// TIA Portal V20 export
TYPE "typeSequenceControlNode"
// stored: Namespace Unit1.Em12
   STRUCT
      jobs : "LAF_typeJobs";
      sequence : "LAF_typeSequence";
      selectJobStatus { S7_SetPoint := 'True'} : Array[0..10] of "LAF_typeJobStatus";
      "step" : "LER_typeStep";
      jobInterface : "Unit1.Em12.typeSequenceControlNodeJobInterface";
      homeCheck : "Unit1.Em12.typeSequenceControlNodeHomeCheck";
   END_STRUCT;
   // // "step".action1[101] : Step[101] : JOB[1] Condition
   // // "step".action1[110] : Step[110] : Clamp Z Up
   // // "step".action1[120] : Step[120] : Clamp Left, Right Open
   // // "step".action1[130] : Step[130] : Clamp Mover Open
   // // "step".action1[180] : Step[180] : Lift Down
   // // "step".action1[190] : Step[190] : JOB[1] Step End
   // // "step".action1[201] : Step[201] : JOB[2] Condition
   // // "step".action1[210] : Step[210] : Stack NG Box [Loading Request] => JR Unloading P&P
   // // "step".action1[220] : Step[220] : Clamp Mover Close
   // // "step".action1[230] : Step[230] : Clamp Left, Right Close
   // // "step".action1[231] : Step[231] : Stack NG Box [Loading Ready] => JR Unloading P&P
   // // "step".action1[290] : Step[290] : JOB[2] Step End
   // // "step".action1[301] : Step[301] : JOB[3] Condition
   // // "step".action1[310] : Step[310] : Clamp Z Down
   // // "step".action1[320] : Step[320] : Clamp Left, Right Open
   // // "step".action1[330] : Step[330] : Clamp Mover Open
   // // "step".action1[340] : Step[340] : Clamp Z Up
   // // "step".action1[390] : Step[390] : JOB[3] Step End
   // // "step".transition1[101] : Step[101] : JOB[1] Condition
   // // "step".transition1[110] : Step[110] : Clamp Z Up
   // // "step".transition1[120] : Step[120] : Clamp Left, Right Open
   // // "step".transition1[130] : Step[130] : Clamp Mover Open
   // // "step".transition1[180] : Step[180] : Lift Down
   // // "step".transition1[190] : Step[190] : JOB[1] Step End
   // // "step".transition1[201] : Step[201] : JOB[2] Condition
   // // "step".transition1[210] : Step[210] : Stack NG Box [Loading Request] => JR Unloading P&P
   // // "step".transition1[220] : Step[220] : Clamp Mover Close
   // // "step".transition1[230] : Step[230] : Clamp Left, Right Close
   // // "step".transition1[231] : Step[231] : Stack NG Box [Loading Ready] => JR Unloading P&P
   // // "step".transition1[290] : Step[290] : JOB[2] Step End
   // // "step".transition1[301] : Step[301] : JOB[3] Condition
   // // "step".transition1[310] : Step[310] : Clamp Z Down
   // // "step".transition1[320] : Step[320] : Clamp Left, Right Open
   // // "step".transition1[330] : Step[330] : Clamp Mover Open
   // // "step".transition1[340] : Step[340] : Clamp Z Up
   // // "step".transition1[390] : Step[390] : JOB[3] Step End
END_TYPE
